// TIA Portal V20 export
ORGANIZATION_BLOCK "Diagnostic error interrupt"   // OB82, FBD, DiagnosticErrorInterrupt
{ S7_Optimized_Access := 'TRUE' }
// stored: SetENOAutomatically false
   VAR_INPUT
      IO_State : Word;   // IO state of the HW object
      LADDR : HW_ANY;   // Hardware identifier
      Channel : UInt;   // Channel number
      MultiError : Bool;   // =true if more than one error is present
   END_VAR
BEGIN

NETWORK
TITLE = call diagnose
      CALL  "Diag", "Diag_DB";

END_ORGANIZATION_BLOCK
